(* CoDeSys 2.3 export: FUNCPARAMS_TS.EXP *)

(* Data type in Diag/Other *)
TYPE FuncParams_ts :
STRUCT
	Description_as8		: STRING(32);
(*	Description_as8		: ARRAY [1..4] OF STRING(32);*)
END_STRUCT
END_TYPE
